Fanuc KAREL source: kb00002.KL

PROGRAM KB00002
%STACKSIZE=65535
%PRIORITY=65535
%NOLOCKGROUP
VAR
P1 : INTEGER
RESULT : INTEGER
BEGIN
P1=1
-- UNRESOLVED_PC line 8 opcodes [21 50 23] marker_code=12
END KB00002
